Yaskawa INFORM job: JERIKAN4.JBI

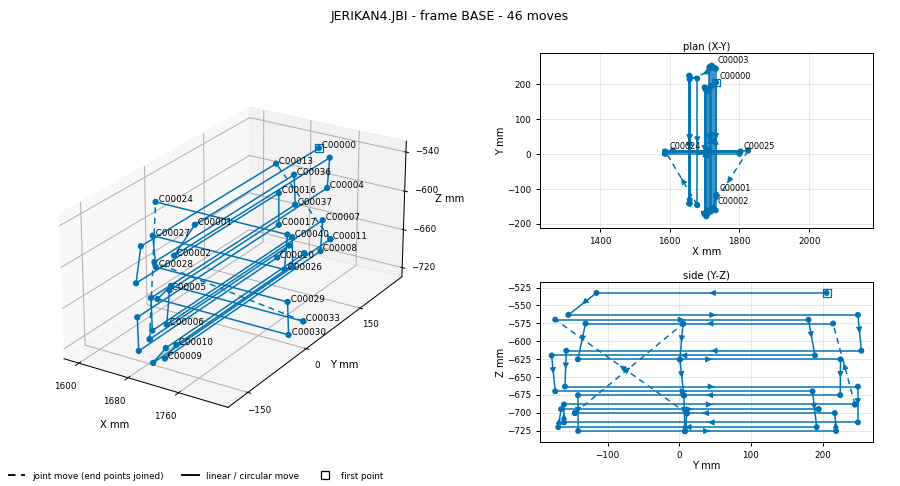
[picture p0: tool path of JERIKAN4.JBI in frame BASE, 46 of 52 moves have a stored position in this frame; points joined in program order, loops and branches not executed]
/JOB
//NAME JERIKAN4
//POS
///NPOS 46,0,46,0,0,0
///TOOL 0
///POSTYPE BASE
///RECTAN
///RCONF 1,0,0,0,0,0,0,0,0,0,0,0,0,0,0,0,0,0,0,0,0,0,0,0
C00000=1733.303989,205.597005,-532.552749,175.000000,-89.999999,5.000000
C00001=1733.303989,-115.703683,-532.552749,175.000000,-89.999999,5.000000
C00002=1726.488085,-154.871410,-563.237154,175.000000,-89.999999,5.000000
C00003=1726.488085,249.265145,-563.237154,175.000000,-89.999999,5.000000
C00004=1720.415612,254.117133,-613.237154,175.000000,-89.999999,5.000000
C00005=1720.415612,-157.753720,-613.237154,175.000000,-89.999999,5.000000
C00006=1716.537865,-159.580693,-663.237154,175.000000,-89.999999,5.000000
C00007=1716.537865,249.265145,-663.237154,175.000000,-89.999999,5.000000
C00008=1713.658839,249.265145,-713.237154,175.000000,-89.999999,5.000000
C00009=1713.658839,-160.988705,-713.237154,175.000000,-89.999999,5.000000
C00010=1732.257607,-160.988705,-688.237154,180.000000,-60.000000,0.000000
C00011=1732.257607,245.217874,-688.237154,180.000000,-60.000000,0.000000
C00012=1732.257607,245.217874,-688.237154,180.000000,-60.000000,0.000000
C00013=1657.676025,214.575039,-575.223120,175.000000,-89.999999,5.000000
C00014=1657.676025,-130.908152,-575.223120,175.000000,-89.999999,5.000000
C00015=1656.251389,-141.552982,-625.223120,175.000000,-89.999999,5.000000
C00016=1656.251389,225.026003,-625.223120,175.000000,-89.999999,5.000000
C00017=1656.983401,224.626534,-675.223120,175.000000,-89.999999,5.000000
C00018=1656.983401,-141.366371,-675.223120,175.000000,-89.999999,5.000000
C00019=1658.026619,-141.202380,-725.223120,175.000000,-89.999999,5.000000
C00020=1658.026619,218.908917,-725.223120,175.000000,-89.999999,5.000000
C00021=1679.272822,217.105864,-700.223120,180.000000,-60.000000,0.000000
C00022=1679.272822,-145.737593,-700.223120,180.000000,-60.000000,0.000000
C00023=1679.272822,-145.737593,-700.223120,180.000000,-60.000000,0.000000
C00024=1589.444892,5.193953,-575.528917,175.000000,-89.999999,5.000000
C00025=1801.670102,5.193953,-575.528917,175.000000,-89.999999,5.000000
C00026=1800.339604,0.815485,-625.528917,175.000000,-89.999999,5.000000
C00027=1586.619587,0.815485,-625.528917,175.000000,-89.999999,5.000000
C00028=1587.194677,6.398614,-675.528917,175.000000,-89.999999,5.000000
C00029=1802.248393,6.398614,-675.528917,175.000000,-89.999999,5.000000
C00030=1803.464726,7.880328,-725.528917,175.000000,-89.999999,5.000000
C00031=1587.947950,7.880328,-725.528917,175.000000,-89.999999,5.000000
C00032=1609.643510,10.538480,-700.528917,180.000000,-60.000000,0.000000
C00033=1824.892479,10.538480,-700.528917,180.000000,-60.000000,0.000000
C00034=1824.892479,10.538480,-700.528917,180.000000,-60.000000,0.000000
C00035=1707.934989,-173.167374,-569.841329,175.000000,-89.999999,5.000000
C00036=1707.934989,180.309255,-569.841329,175.000000,-89.999999,5.000000
C00037=1705.082708,189.342872,-619.841329,175.000000,-89.999999,5.000000
C00038=1705.082708,-178.178451,-619.841329,175.000000,-89.999999,5.000000
C00039=1702.734351,-173.196662,-669.841329,175.000000,-89.999999,5.000000
C00040=1702.734351,185.996037,-669.841329,175.000000,-89.999999,5.000000
C00041=1700.273500,191.745448,-719.841329,175.000000,-89.999999,5.000000
C00042=1700.273500,-168.973374,-719.841329,175.000000,-89.999999,5.000000
C00043=1718.123414,-164.928428,-694.841329,180.000000,-60.000000,0.000000
C00044=1718.123414,194.418926,-694.841329,180.000000,-60.000000,0.000000
C00045=1718.123414,194.418926,-694.841329,180.000000,-60.000000,0.000000
///POSTYPE PULSE
///PULSE
EC00000=0
EC00001=0
EC00002=0
EC00003=0
EC00004=0
EC00005=0
EC00006=0
EC00007=0
EC00008=0
EC00009=0
EC00010=0
EC00011=0
EC00012=92160
EC00013=92160
EC00014=92160
EC00015=92160
EC00016=92160
EC00017=92160
EC00018=92160
EC00019=92160
EC00020=92160
EC00021=92160
EC00022=92160
EC00023=184320
EC00024=184320
EC00025=184320
EC00026=184320
EC00027=184320
EC00028=184320
EC00029=184320
EC00030=184320
EC00031=184320
EC00032=184320
EC00033=184320
EC00034=276480
EC00035=276480
EC00036=276480
EC00037=276480
EC00038=276480
EC00039=276480
EC00040=276480
EC00041=276480
EC00042=276480
EC00043=276480
EC00044=276480
EC00045=368640
//INST
///DATE 2023/02/08 11:05
///ATTR SC,RW,RJ
////FRAME BASE
///GROUP1 RB1,ST1
NOP
MOVJ P009 EX000 VJ=15.00
MOVJ P009 VJ=15.00
MOVJ C00000 EC00000 VJ=15.0
CALL JOB:SPYON
MOVL C00001 EC00001 V=150.0
MOVL C00002 EC00002 V=150.0
MOVL C00003 EC00003 V=150.0
MOVL C00004 EC00004 V=150.0
MOVL C00005 EC00005 V=150.0
MOVL C00006 EC00006 V=150.0
MOVL C00007 EC00007 V=150.0
MOVL C00008 EC00008 V=150.0
MOVL C00009 EC00009 V=150.0
MOVL C00010 EC00010 V=150.0
MOVL C00011 EC00011 V=150.0
CALL JOB:SPYOF
MOVJ P009 VJ=15.00
MOVL C00012 EC00012 V=150.0
MOVJ C00013 EC00013 VJ=15.0
CALL JOB:SPYON
MOVL C00014 EC00014 V=150.0
MOVL C00015 EC00015 V=150.0
MOVL C00016 EC00016 V=150.0
MOVL C00017 EC00017 V=150.0
MOVL C00018 EC00018 V=150.0
MOVL C00019 EC00019 V=150.0
MOVL C00020 EC00020 V=150.0
MOVL C00021 EC00021 V=150.0
MOVL C00022 EC00022 V=150.0
CALL JOB:SPYOF
MOVJ P009 VJ=15.00
MOVL C00023 EC00023 V=150.0
MOVJ C00024 EC00024 VJ=15.0
CALL JOB:SPYON
MOVL C00025 EC00025 V=150.0
MOVL C00026 EC00026 V=150.0
MOVL C00027 EC00027 V=150.0
MOVL C00028 EC00028 V=150.0
MOVL C00029 EC00029 V=150.0
MOVL C00030 EC00030 V=150.0
MOVL C00031 EC00031 V=150.0
MOVL C00032 EC00032 V=150.0
MOVL C00033 EC00033 V=150.0
CALL JOB:SPYOF
MOVJ P009 VJ=15.00
MOVL C00034 EC00034 V=150.0
MOVJ C00035 EC00035 VJ=15.0
CALL JOB:SPYON
MOVL C00036 EC00036 V=150.0
MOVL C00037 EC00037 V=150.0
MOVL C00038 EC00038 V=150.0
MOVL C00039 EC00039 V=150.0
MOVL C00040 EC00040 V=150.0
MOVL C00041 EC00041 V=150.0
MOVL C00042 EC00042 V=150.0
MOVL C00043 EC00043 V=150.0
MOVL C00044 EC00044 V=150.0
CALL JOB:SPYOF
MOVJ P009 VJ=15.00
MOVL C00045 EC00045 V=150.0
END
